TYPE ST_WorkTime :
STRUCT
	Hours	: UDINT; 
	Minutes : UINT;	 	
	Seconds	: UINT;
	Display : T_MaxString; // formatowany string np 12:35:06
	Running	: BOOL;		   // informacja pomocnicza czy aktualnie trwa zliczanie	
 
END_STRUCT
END_TYPE

(* stored: Version 1.1.0.1, ProductVersion 3.1.4024.15
   DUT ST_WorkTime: Id {759e6b42-10ff-4fce-9501-21df78544ed2} *)
